PROGRAM z_FILL


(*-------------------------------------------------------------------------------------------------------*)
(*v001  Llenado agua fria*)
Mc._04_FILL.v001_Cool.xOpen:= F_LLENADO.z_xCWater OR
							F_LAVADO_CONT.z_xAguaFria;

(*-------------------------------------------------------------------------------------------------------*)
(*v002  Llenado agua Caliente*)
Mc._04_FILL.v002_Hot.xOpen := F_LLENADO.z_xHWater OR 
							F_LAVADO_CONT.z_xAguaCaliente;

(*-------------------------------------------------------------------------------------------------------*)
(*v003  Hard Water Fill*)
Mc._04_FILL.v003_Hard.xOpen:= F_LLENADO.z_xHWater OR
							F_LAVADO_CONT.z_xAguaDura;

(*-------------------------------------------------------------------------------------------------------*)
(*v005  Llenado Salmuera*)

(*-------------------------------------------------------------------------------------------------------*)
(*v006  Intercepta Llenado*)
Mc._04_FILL.v006_InterMc.xOpen:= F_LLENADO.xFillInterceptValve;

END_PROGRAM

(* stored: Version 1.1.0.1, ProductVersion 3.1.4024.10
   POU z_FILL: Id {05b7e967-6f4f-4a41-b973-30add8500adf}, SpecialFunc None *)
